// TIA Portal V19 export
TYPE "MotorSts"
// stored: Access Published
   STRUCT
      AlarmPresence : Bool;   // Cumulative alarm presence
      RunPermitted : Bool;   // Motor run permitted
      Running : Bool;   // State of motor running / Motor running
   END_STRUCT;
END_TYPE
